// TwinCAT 3 PLC project Untitled1
// ProgramVersion: 3.1.4024.0
// libraries:
//   Tc2_Standard, * (Beckhoff Automation GmbH)
//   Tc2_System, * (Beckhoff Automation GmbH)
//   Tc3_Module, * (Beckhoff Automation GmbH)
//   VisuSymbols,3.5.10.0,System
// project tree:
//   / GlobalTextList.TcGTLO, PlcTask.TcTTO, Task_1.TcTTO, Task_2.TcTTO, Visualization Manager.TcVMO (not stored)
//   POUs/ CarTrafficLight.TcPOU, Function_SettingCarLight.TcPOU, Function_SettingPedestrianLight.TcPOU, GVL.TcGVL, MAIN.TcPOU, PedestrianTrafficLight.TcPOU, Visualization_Trafficlight_system.TcVIS
//   VISUs/ Visualization_Trafficlight.TcVIS
// real-time tasks:
//   TASK PlcTask: cycle T#10ms, priority 20, ADS port 350
//   TASK Task 1: cycle T#10ms, priority 1, ADS port 351
//   TASK Task 2: cycle T#10ms, priority 2, ADS port 352

CONFIGURATION Untitled1
    RESOURCE PLC ON TwinCAT3
        TASK PlcTask(INTERVAL := T#10ms, PRIORITY := 20);
        TASK Task_1(INTERVAL := T#10ms, PRIORITY := 1);
        TASK Task_2(INTERVAL := T#10ms, PRIORITY := 2);
        PROGRAM MAIN WITH PlcTask : MAIN;
        PROGRAM CarTrafficLight WITH Task_1 : CarTrafficLight;
        PROGRAM PedestrianTrafficLight WITH Task_2 : PedestrianTrafficLight;
    END_RESOURCE
END_CONFIGURATION

// ---- POUs/GVL.TcGVL
{attribute 'qualified_only'}
VAR_GLOBAL
	
// Car light status
CarLightRed : BOOL := FALSE;
CarLightYellow : BOOL := FALSE;
CarLightGreen : BOOL := TRUE;

// Timers for transitions
TONCarGreenToYellow : TON;
TONCarYellowToRed : TON;
TONCarRedToGreen : TON;
TONPedestrianGreen : TON;

// Pedestrian light status
PedestrianLightRed : BOOL := TRUE;
PedestrianLightGreen : BOOL := FALSE;

// Detects if there is a person to cross the road
ButtonPedestrian : BOOL := FALSE;
CarSensor : BOOL := FALSE;

// Status traffic lights
StatusCarLight : INT := 0;
StatusPedestrianLight : INT := 0;

//Blinker Pedestrian traffic light
TONBlinkerTimer : TON;

	
END_VAR

// ---- POUs/MAIN.TcPOU
PROGRAM MAIN
VAR


END_VAR

CarTrafficLight();
PedestrianTrafficLight();

END_PROGRAM

// ---- POUs/CarTrafficLight.TcPOU
PROGRAM CarTrafficLight
VAR

	GreenToYellowTimerOn : BOOL := FALSE;
    YellowToRedTimerOn : BOOL := FALSE;
    RedToGreenTimerOn : BOOL := FALSE;
END_VAR

CASE GVL.StatusCarLight OF
	
//Green light
0: IF GVL.ButtonPedestrian THEN
	GVL.StatusCarLight := 3;
   ELSE
   Function_SettingCarLight(2);
   END_IF
   
//Yellow Light
1:  Function_SettingCarLight (1);
	            
	GVL.TONCarYellowToRed ( IN := TRUE , PT := T#3S);  //Start timer to go to red light
          
	    IF GVL.TONCarYellowToRed.Q THEN        // If timer reaches 3s traffic light turns red
		   GVL.StatusCarLight := 2;
		   GVL.TONCarYellowToRed ( IN := FALSE);
       END_IF
	   
//Red Light
2: IF GVL.CarSensor THEN
     GVL.StatusCarLight :=4;
   ELSE
     Function_SettingCarLight (0);
   END_IF 
	  
//Waiting time green to yellow
3: GVL.TONCarGreenToYellow (IN := TRUE , PT := T#10s);
   IF GVL.TONCarGreenToYellow.Q THEN
      GVL.StatusCarLight := 1;
	  GVL.TONCarGreenToYellow (IN := FALSE);
   END_IF	

// Waiting time Red to Green
4: GVL.TONCarRedToGreen ( IN := TRUE, PT := T#10S);   //Start timer to go to green light
          
   IF GVL.TONCarRedToGreen.Q THEN        // If timer reaches 10s traffic light turns green
	  GVL.StatusCarLight := 0;
	  GVL.TONCarRedToGreen ( IN := FALSE);
   END_IF
END_CASE

END_PROGRAM

// ---- POUs/Function_SettingCarLight.TcPOU
FUNCTION Function_SettingCarLight : BOOL
VAR_INPUT
	ColorCarLight : INT; // 0 for Red, 1 for Green
    
END_VAR
VAR
END_VAR

// Set the light state
CASE ColorCarLight OF
    0:  // Red
        GVl.PedestrianLightRed := TRUE;
        GVL.PedestrianLightGreen := FALSE;
    
    1:  // Green
        GVL.PedestrianLightRed := FALSE;
        GVL.PedestrianLightGreen := TRUE;
END_CASE;

Function_SettingPedestrianLight := TRUE;

END_FUNCTION

// ---- POUs/Function_SettingPedestrianLight.TcPOU
FUNCTION Function_SettingPedestrianLight : BOOL
VAR_INPUT
	ColorPedestrianLight : INT; // 0 for Red, 1 for Yellow, 2 for Green
END_VAR
VAR
END_VAR

// Set the light state 
CASE ColorPedestrianLight OF
    0:  // Red
        GVl.CarLightRed := TRUE;
        GVL.CarLightYellow := FALSE;
        GVL.CarLightGreen := FALSE;
    1:  // Yellow
        GVL.CarLightRed := FALSE;
        GVL.CarLightYellow := TRUE;
        GVL.CarLightGreen := FALSE;
    2:  // Green
        GVL.CarLightRed := FALSE;
        GVL.CarLightYellow := FALSE;
        GVL.CarLightGreen := TRUE;
END_CASE;

Function_SettingCarLight := TRUE;

END_FUNCTION

// ---- POUs/PedestrianTrafficLight.TcPOU
PROGRAM PedestrianTrafficLight
VAR
	GreenTimerOn : BOOL := FALSE;
END_VAR

CASE GVL.StatusPedestrianLight OF

//Red Light
   0:
      Function_SettingPedestrianLight (0);
	  
	  IF GVL.StatusCarLight = 2 THEN
		 GVL.StatusPedestrianLight := 1;
	  END_IF
	  
//Green light
   1:IF GVL.CarSensor THEN
	   GVL.StatusPedestrianLight := 2;
     ELSE
     Function_SettingPedestrianLight (1);
	 END_IF
	 
// Waiting time for car	 
2:  GVL.TONPedestrianGreen(IN := TRUE , PT := T#10S);
	
    IF GVL.TONPedestrianGreen.ET >= T#5S THEN
       GVL.TONBlinkerTimer (IN := TRUE , PT := T#500MS );
       IF GVL.TONBlinkerTimer.Q THEN
          GVL.PedestrianLightGreen := NOT GVL.PedestrianLightGreen;
		  GVL.TONBlinkerTimer (IN := FALSE);
		  GVL.TONBlinkerTimer (IN := TRUE);
	   END_IF
	ELSE
		GVL.PedestrianLightGreen := TRUE;
    END_IF
	
    IF GVL.TONPedestrianGreen.Q THEN
	   GVL.StatusPedestrianLight := 0;
       GVL.TONPedestrianGreen (IN := FALSE);
	   GVL.TONBlinkerTimer (IN := FALSE);
	   GVL.PedestrianLightGreen := FALSE;
	END_IF
END_CASE

END_PROGRAM

// ---- GlobalTextList.TcGTLO
TEXTLIST GlobalTextList
  242 = 'Car Sensor'
  854 = 'Pedestrian'
  620 = 'Pedestrian button'
  314 = 'Pedestrian Button'
  370 = 'Pedestrian Light'
  261 = 'Pedestrian Sensor'
  570 = 'Pedestrian Switch'
  378 = 'Traffic'
  988 = 'Traffic light'
  852 = 'Traffic Sensor'
END_TEXTLIST

// ---- POUs/Visualization_Trafficlight_system.TcVIS
VISUALIZATION Visualization_Trafficlight_system  // 2x2
END_VISUALIZATION

// ---- VISUs/Visualization_Trafficlight.TcVIS
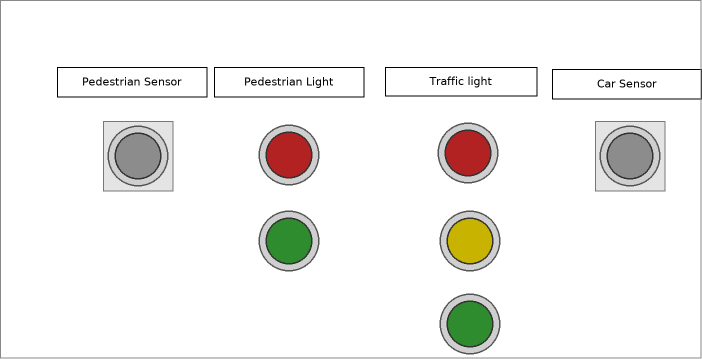
VISUALIZATION Visualization_Trafficlight  // 702x359
    Lamp1 (433,118 70x70), variable: GVL.CarLightRed, style: Lamp-Lamp1-Red
    Lamp1 (435,206 70x70), variable: GVL.CarLightYellow, style: Lamp-Lamp1-Yellow
    Lamp1 (435,289 70x70), variable: GVL.CarLightGreen, style: Lamp-Lamp1-Green
    Rectangle (385,67 152x29), "Traffic light"
    Rectangle (57,67 150x30), "Pedestrian Sensor"
    Lamp1 (254,120 70x70), variable: GVL.PedestrianLightRed, style: Lamp-Lamp1-Red
    Lamp1 (254,206 70x70), variable: GVL.PedestrianLightGreen, style: Lamp-Lamp1-Green
    Rectangle (214,67 150x30), "Pedestrian Light"
    PushSwitch (103,121 70x70), variable: GVL.ButtonPedestrian, behaviour: TOGGLE, style: Switch-PushSwitch-Gray
    PushSwitch (595,121 70x70), variable: GVL.CarSensor, behaviour: TOGGLE, style: Switch-PushSwitch-Gray
    Rectangle (552,69 150x30), "Car Sensor"
END_VISUALIZATION
